Xinje XDPPro project, PLC1: XD5-48T6 (software 3.7.4b 2021-06-17)

PROGRAM Ladder

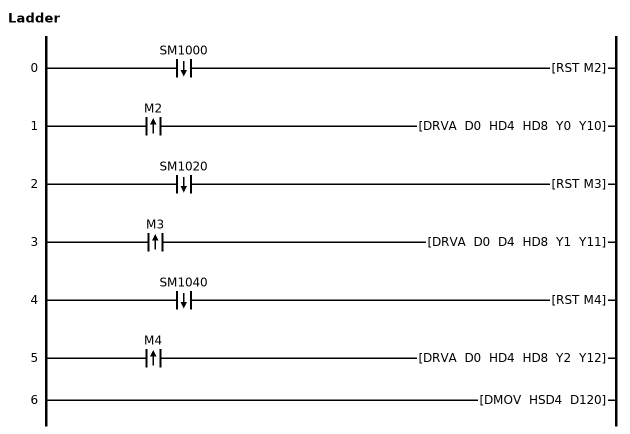
LDF    SM1000
RST    M2
LDP    M2
DRVA   D0 HD4 HD8 Y0 Y10
LDF    SM1020
RST    M3
LDP    M3
DRVA   D0 D4 HD8 Y1 Y11
LDF    SM1040
RST    M4
LDP    M4
DRVA   D0 HD4 HD8 Y2 Y12
DMOV   HSD4 D120